# EPICS alarm handler configuration: alh_files/mgnt_in20Ilhe_soln.alhConfig
GROUP NULL SOLN:IN20ILHE:MG01
   $COMMAND edm -x -eolc -noedit mgnt_in20_soln.edl
$ALIAS SOLN
$GUIDANCE
IN20ILHE soln magnets
   Group Name: SOLN:IN20ILHE:MG01
   Summary PV:  SOLN:IN20ILHE:MG01:STATSUMY
$END

GROUP SOLN:IN20ILHE:MG01  SOLN:IN20:311
   $COMMAND edm -x -eolc -noedit -m "DEV=SOLN:IN20:311" mgnt_unit.edl
CHANNEL   SOLN:IN20:311       SOLN:IN20:311:STATMSG                 ----L
   $FORCEPV SOLN:IN20:311:STATMSGSV -DATL 1 0
